PROGRAM P_Iterator
VAR
    Notifications 	: NotificationCollection;
	n			: Object;
	iterator	  	: Iterator;

	bInit			: BOOL;
	bReset			: BOOL;
END_VAR

IF NOT bInit THEN
	bInit := TRUE;
	
	Notifications.addItem(str := 'The');
	Notifications.addItem(str := 'quick');
	Notifications.addItem(str := 'brown');
	Notifications.addItem(str := 'fox');
	Notifications.addItem(str := 'jumps');
	Notifications.addItem(str := 'over');
	Notifications.addItem(str := 'the');
	Notifications.addItem(str := 'lazy');
	Notifications.addItem(str := 'dog');
	
	iterator := notifications.createIterator();	
	n := Iterator.current();
	F_VerboseLogger(n.getNotification());
END_IF




WHILE(Iterator.hasNext()) DO
	n := Iterator.next();
	F_VerboseLogger(n.getNotification());
END_WHILE

IF bReset THEN
	iterator.reset();
	n := Iterator.current();
	F_VerboseLogger(n.getNotification());
	bReset := FALSE;
END_IF

END_PROGRAM

(* stored: Version 1.1.0.1, ProductVersion 3.1.4024.12
   POU P_Iterator: Id {e6f2f43d-3006-4b61-a734-eb841ad749f8}, SpecialFunc None *)
